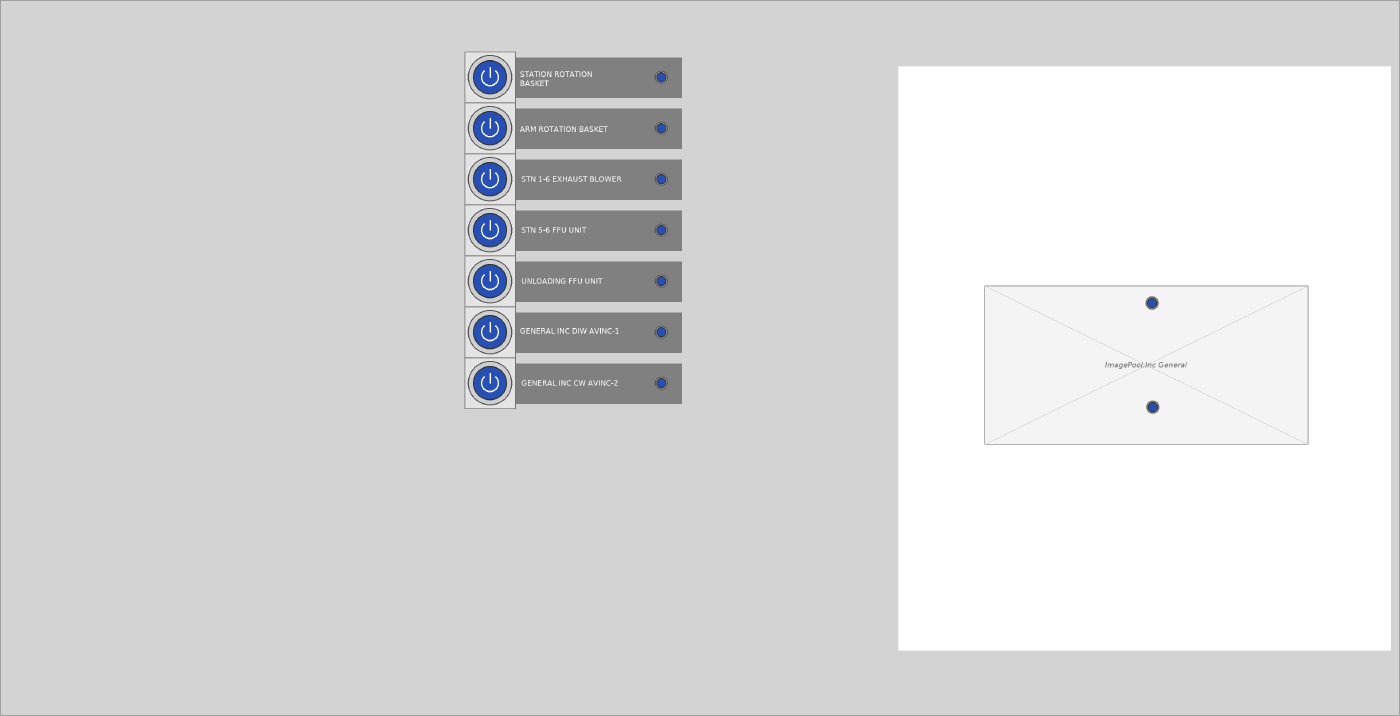
VISUALIZATION Manual_General  // 1920x983
    Rectangle (0,0 1920x983)
    Rectangle (1232,91 675x802)
    Image (1350,392 444x218), image: ImagePool.Inc General
    RoundedRectangle (676,79 259x55)
    Label (710,94 176x29), "STATION ROTATION BASKET"
    Lamp1 (897,96 20x20), variable: ARdsMAP_HmiVariableGeneral.bStnRotationRotaryBarrel_IND, style: Lamp-Lamp1-Blue
    PowerSwitch (637,71 70x70), variable: ARdsMAP_HmiVariableGeneral.bStnRotationRotaryBarrel_PB, behaviour: TOGGLE, style: Switch-PowerSwitch-Blue
    RoundedRectangle (676,149 259x55)
    Label (710,160 177x35), "ARM ROTATION BASKET"
    Lamp1 (897,166 20x20), variable: ARdsMAP_HmiVariableGeneral.bRobotRotationRotaryBarrel_IND, style: Lamp-Lamp1-Blue
    PowerSwitch (637,141 70x70), variable: ARdsMAP_HmiVariableGeneral.bRobotRotationRotaryBarrel_PB, behaviour: TOGGLE, style: Switch-PowerSwitch-Blue
    RoundedRectangle (676,219 259x55)
    Label (712,228 160x36), "STN 1-6 EXHAUST BLOWER"
    Lamp1 (897,236 20x20), variable: ARdsMAP_HmiVariableGeneral.bExhaustBlower_IND, style: Lamp-Lamp1-Blue
    PowerSwitch (637,211 70x70), variable: ARdsMAP_HmiVariableGeneral.bExhaustBlower_PB, behaviour: TOGGLE, style: Switch-PowerSwitch-Blue
    RoundedRectangle (676,429 259x55)
    Label (710,440 178x29), "GENERAL INC DIW AVINC-1"
    Lamp1 (897,446 20x20), variable: ARdsMAP_HmiVariableGeneral.bGeneralIncValve01_IND, style: Lamp-Lamp1-Blue
    PowerSwitch (637,421 70x70), variable: ARdsMAP_HmiVariableGeneral.bGeneralIncValve01_PB, behaviour: TOGGLE, style: Switch-PowerSwitch-Blue
    RoundedRectangle (676,499 259x55)
    Label (712,508 189x36), "GENERAL INC CW AVINC-2"
    Lamp1 (897,516 20x20), variable: ARdsMAP_HmiVariableGeneral.bGeneralIncValve02_IND, style: Lamp-Lamp1-Blue
    PowerSwitch (637,491 70x70), variable: ARdsMAP_HmiVariableGeneral.bGeneralIncValve02_PB, behaviour: TOGGLE, style: Switch-PowerSwitch-Blue
    Lamp1 (1570,406 20x20), variable: ARdsMAP_HmiVariableGeneral.bGeneralIncValve01_IND, style: Lamp-Lamp1-Blue
    Lamp1 (1571,549 20x20), variable: ARdsMAP_HmiVariableGeneral.bGeneralIncValve02_IND, style: Lamp-Lamp1-Blue
    RoundedRectangle (676,289 259x55)
    Label (712,298 160x36), "STN 5-6 FFU UNIT"
    Lamp1 (897,306 20x20), variable: ARdsMAP_HmiVariableGeneral.bFFU01_IND, style: Lamp-Lamp1-Blue
    PowerSwitch (637,281 70x70), variable: ARdsMAP_HmiVariableGeneral.bFFU01_PB, behaviour: TOGGLE, style: Switch-PowerSwitch-Blue
    RoundedRectangle (676,359 259x55)
    Label (712,368 160x36), "UNLOADING FFU UNIT"
    Lamp1 (897,376 20x20), variable: ARdsMAP_HmiVariableGeneral.bFFU02_IND, style: Lamp-Lamp1-Blue
    PowerSwitch (637,351 70x70), variable: ARdsMAP_HmiVariableGeneral.bFFU02_PB, behaviour: TOGGLE, style: Switch-PowerSwitch-Blue
END_VISUALIZATION

(* stored: Version 1.1.0.1, ProductVersion 3.1.4024.12
   Visu Manual_General: Id {ad575fc0-f186-4fa8-9fe9-a966ef3681eb} *)
